TYPE FLOWMETER_CONTROL :
STRUCT

	SET_TOT: USINT;
	SET_MODE: USINT;

END_STRUCT
END_TYPE

(* stored: Version 1.1.0.1, ProductVersion 3.1.0.26
   DUT FLOWMETER_CONTROL: Id {2b4e2f6a-728d-44fa-8d18-fa702140e23a} *)
